FUNCTION_BLOCK TrkEclipse (* Service Interface Function Block Type *)
  (* Standard: 61499-2 *)
  (* Version 0.0, 2012-05-22, 4DIAC-IDE, 4DIAC-Consortium *)
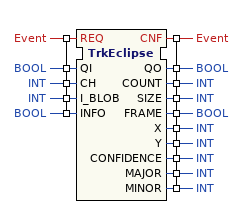
  EVENT_INPUT
    REQ WITH QI, CH, I_BLOB, INFO; (* track_update and returns all information *)
  END_EVENT
  EVENT_OUTPUT
    CNF WITH QO, COUNT, SIZE, FRAME, CONFIDENCE, MAJOR, MINOR, X, Y; (* Confirmation of Requested Service *)
  END_EVENT
  VAR_INPUT
    QI : BOOL; (* Event Input Qualifier *)
    CH : INT; (* channel (0-3) *)
    I_BLOB : INT; (* index of Blob, where 0 is the largest and default, Up to 9 blobs channels supported *)
    INFO : BOOL; (* prints outputs if true=1 *)
  END_VAR
  VAR_OUTPUT
    QO : BOOL; (* Event Output Qualifier *)
    COUNT : INT; (* Number of blobs on a channel. *)
    SIZE : INT; (* size of blob from channel CH and INDEX in pixels *)
    FRAME : BOOL; (* frame number used to generate the tracking data *)
    X : INT; (* X Blob Center *)
    Y : INT; (* Y Blob Center *)
    CONFIDENCE : INT; (* % confidence for seeing the blob in pixel area/bounding box area for CH/INDEX *)
    MAJOR : INT; (* length in pixels of the major axis of the bounding ECLIPSE for the blob from CH/INDEX *)
    MINOR : INT; (* length in pixels of the minor axis of the bounding ECLIPSE for the blob from CH/INDEX *)
  END_VAR
  SERVICE APPLICATION/RESOURCE (* Service Interface Function Block Type *)
    SEQUENCE normal_establishment
      APPLICATION.INIT+(PARAMS) -> APPLICATION.INITO+(PARAMS);
    END_SEQUENCE
    SEQUENCE unsuccessful_establishment
      APPLICATION.INIT+(PARAMS) -> APPLICATION.INITO-(STATUS);
    END_SEQUENCE
    SEQUENCE request_confirm
      APPLICATION.REQ+(SD) -> APPLICATION.CNF+(RD);
    END_SEQUENCE
    SEQUENCE request_inhibited
      APPLICATION.REQ-(SD) -> APPLICATION.CNF-(STATUS);
    END_SEQUENCE
    SEQUENCE request_error
      APPLICATION.REQ+(SD) -> APPLICATION.CNF-(STATUS);
    END_SEQUENCE
    SEQUENCE indication_response
      RESOURCE.indicate(RD) -> APPLICATION.IND+(RD);
      APPLICATION.RSP(QI,SD) -> RESOURCE.response(QI,SD);
    END_SEQUENCE
    SEQUENCE indication_inhibited
      RESOURCE.indicate(RD,QI=FALSE) -> RESOURCE.inhibited();
    END_SEQUENCE
    SEQUENCE error_indication
      RESOURCE.error(STATUS) -> APPLICATION.IND-(STATUS);
    END_SEQUENCE
    SEQUENCE application_initiated_termination
      APPLICATION.INIT-() -> APPLICATION.INITO-(STATUS);
    END_SEQUENCE
    SEQUENCE resource_initiated_termination
      -> APPLICATION.INITO-(STATUS);
    END_SEQUENCE
  END_SERVICE
END_FUNCTION_BLOCK
